Staubli VAL3: insert_cCount.pgx

public program insert_cCount(string x_sItem (dimensions=1), bool x_bActive (dimensions=1), num x_num (dimensions=1))
begin
  // insert a new IO
  if isDefined(cCount[x_sItem])==false
    insert(cCount[x_sItem])
    cCount[x_sItem].bActive=x_bActive
    cCount[x_sItem].sID=x_sItem
    cCount[x_sItem].sName=x_sItem
    cCount[x_sItem].nCount=x_num
    cCount[x_sItem].bEnable=true
  endIf
end
